Universal Robots PolyScope program: Put_into_box_E-series_UR3.urp

Program Put_into_box_E-series_UR3 (installation=default directory=/programs createdIn=3.0.0.0 lastSavedIn=5.2.0.61336 robotSerialNumber=20185300040)
Calibrated DH parameters: a=[-0.000128, -0.221415, -0.194849, 0.000098, -0.000148, 0]; d=[0.152137, 33.879231, 13.968137, -47.716378, 0.085395, 0.092257]; alpha=[1.57105, 0.003021, -0.001826, 1.571145, -1.57192, 0]; deltaTheta=[0, 0.433042, -0.854582, 0.421536, 0.000002, 0]
Robot Program (runOnlyOnce=true)
  Set NoAction (payload=0 tcpAsCog=true)
  MoveJ speed 50 deg/s, acceleration 100 deg/s^2 (useActiveTCP=false positionType=JointAngles) feature=Base
    Waypoint Home: TCP in base x=-0.556 y=-222.914 z=694.011 mm, rx=0.002 ry=-2.2182 rz=2.2173 rad; joints [0, -90.004, 0, -90.005, 0, 0] deg
    Waypoint End: TCP in base x=-222.255 y=-140.418 z=254.023 mm, rx=1.2057 ry=-1.2004 rz=-1.2169 rad; joints [-90, -180, 152, -242, 0, 270] deg
